// TIA Portal V16 export
// export: Created 2023-01-04T15:44:08.9562795Z, ExportSetting WithDefaults, DisplayName Totally Integrated Automation Portal, DisplayVersion V16, DisplayName TIA Portal Version Control Interface, DisplayVersion V16, DisplayName TIA Portal Openness, DisplayVersion V16, DisplayName STEP 7 Professional, DisplayVersion V16, DisplayName STEP 7 Safety, DisplayVersion V16, DisplayName WinCC Advanced, DisplayVersion V16
FUNCTION_BLOCK "Tank2"   // FB5, LAD
{ S7_Optimized_Access := 'TRUE' }
VERSION : 0.1
// stored: AutoNumber true, IsIECCheckEnabled false, IsRetainMemResEnabled false, MemoryReserve 100, SetENOAutomatically false, UDAEnableTagReadback false
   VAR_INPUT
      EN_2 : Bool;
   END_VAR
   VAR_TEMP   // added for the SCL form of the ladder/FBD networks
      _w1 : Bool;
      _w2 : Bool;
      _w3 : Bool;
   END_VAR
BEGIN

REGION Network 1
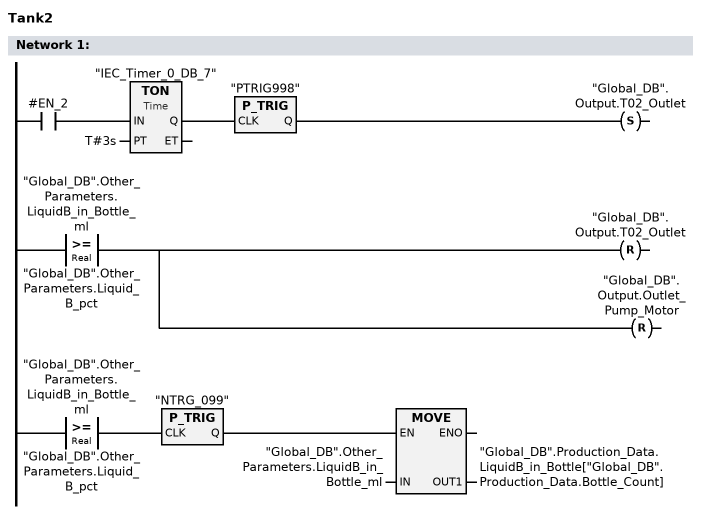
   RUNG wire#powerrail
      Contact( #EN_2 )
      { S7_Templates := "time_type := Time" } "IEC_Timer_0_DB_7".TON(pt := T#3s, et =>)
      P_Trig( "PTRIG998" )
      S_Coil( "Global_DB".Output.T02_Outlet )
   END_RUNG
   RUNG wire#powerrail
      { S7_Templates := "SrcType := Real" } GE_Contact(in1 := "Global_DB".Other_Parameters.LiquidB_in_Bottle_ml, in2 := "Global_DB".Other_Parameters.Liquid_B_pct)
      wire#w1
      R_Coil( "Global_DB".Output.T02_Outlet )
   END_RUNG
   RUNG wire#w1
      R_Coil( "Global_DB".Output.Outlet_Pump_Motor )
   END_RUNG
   RUNG wire#powerrail
      { S7_Templates := "SrcType := Real" } GE_Contact(in1 := "Global_DB".Other_Parameters.LiquidB_in_Bottle_ml, in2 := "Global_DB".Other_Parameters.Liquid_B_pct)
      P_Trig( "NTRG_099" )
      Move(in := "Global_DB".Other_Parameters.LiquidB_in_Bottle_ml, out1 => "Global_DB".Production_Data.LiquidB_in_Bottle["Global_DB".Production_Data.Bottle_Count])
   END_RUNG
   // the same network as SCL:
   "IEC_Timer_0_DB_7".TON(IN := #EN_2, PT := T#3s);
   #_w1 := "IEC_Timer_0_DB_7".Q AND NOT "PTRIG998";   // rising edge
   "PTRIG998" := "IEC_Timer_0_DB_7".Q;
   IF #_w1 THEN "Global_DB".Output.T02_Outlet := TRUE; END_IF;
   IF "Global_DB".Other_Parameters.LiquidB_in_Bottle_ml >= "Global_DB".Other_Parameters.Liquid_B_pct THEN
       "Global_DB".Output.T02_Outlet := FALSE;
       "Global_DB".Output.Outlet_Pump_Motor := FALSE;
   END_IF;
   #_w2 := "Global_DB".Other_Parameters.LiquidB_in_Bottle_ml >= "Global_DB".Other_Parameters.Liquid_B_pct;
   #_w3 := #_w2 AND NOT "NTRG_099";   // rising edge
   "NTRG_099" := #_w2;
   IF #_w3 THEN
       "Global_DB".Production_Data.LiquidB_in_Bottle["Global_DB".Production_Data.Bottle_Count] := "Global_DB".Other_Parameters.LiquidB_in_Bottle_ml;
   END_IF;
END_REGION
END_FUNCTION_BLOCK
